// TIA Portal V20 export
TYPE "typeSequenceControlNodeConveyorJobInterfaceMonitoring"
// stored: Namespace Unit1.Em7
   STRUCT
      spare { ExternalWritable := 'False'} : Bool;
   END_STRUCT;
END_TYPE
